(*********************************** G.D S.p.A. - Technical Department ***********************************
============= PROGRAM INFO ============
FOLDER:             TBD
MACHINES INVOLVED:  TBD 

============= DESCRIPTION =============
csp machine declaration

============= REVISIONS ===============
Date		Version	 	Author      	Description             
----------	-------		------------  	--------------------------------------------
2019/04/05 	0000.00	 	M.Grasso		Creation of the PRG

**********************************************************************************************************)
(*$R process_ref := prc; $*)
PROGRAM csp_transfer_infeed_accumulation
VAR
	
	prc:											process;
	prc_path:										STRING;
	
	accumulation_conveyor_running:					BOOL;
	disable_req:									BOOL;
	
	
END_VAR

_read_var_input();

_object_manager();

IF NOT objects_running()
THEN
	RETURN;	
END_IF

_read_process_image();

_mode_manager();

CASE process_get_mode(prc) OF
	MODE_ABSENT,
	MODE_INACTIVE:
		RETURN;
	MODE_TEST:
		_handle_process_test();
END_CASE


_set_runtime_properties();

(********************************* BODY *********************************)
(************************************************************************)

accumulation_conveyor_running := axis_is_moving(csp_transfer_infeed_accumulation_belt.axis);

disable_req := NOT
				((
				csp_transfer_infeed.run_infeed_belts
				)
				AND
				process_is_ready(prc)
				AND
				process_subtree_is_ready(prc));


_handle_messages();

_write_output();

ACTION _handle_messages:
;
END_ACTION

ACTION _handle_process_test:
;
END_ACTION

ACTION _mode_manager:
IF process_mode_req_is_pending(prc)
THEN
    process_apply_mode_req_first_step(prc);
    CASE process_get_mode(prc) OF
        MODE_TO_ABSENT:
			;
        MODE_TO_INACTIVE:
			;
        MODE_TO_TEST:
			;
        MODE_TO_OPERATIONAL:
			;
    END_CASE
    process_apply_mode_req_second_step(prc);
END_IF
END_ACTION

ACTION _object_manager:
IF objects_initialization()
THEN
	sub_process_init(
		object_name					:= 'csp_transfer_infeed_accumulation.prc', 
		process						:= csp_transfer_infeed.prc, 
		CONVERSION_this				:= prc);
		
	prc_path 						:= process_get_path(prc);
	
END_IF

IF objects_running()
THEN
	process_cycle(prc);
END_IF
END_ACTION

ACTION _read_process_image:
;
END_ACTION

ACTION _read_var_input:
;
END_ACTION

ACTION _set_runtime_properties:
;
END_ACTION

ACTION _write_output:
;
END_ACTION

END_PROGRAM

(* stored: Version 1.1.0.1, ProductVersion 3.1.4024.3
   POU csp_transfer_infeed_accumulation: Id {a79cd134-3646-4220-9711-3f94c224ec2d}, SpecialFunc None
   Action _handle_messages: Id {b79f2d6d-428a-4ddf-8301-7fd94ca80f10}
   Action _handle_process_test: Id {f858689f-18b2-4f51-95e1-907e4326fa7a}
   Action _mode_manager: Id {b55a7ea0-3679-46bc-808b-ce3e5b871f1a}
   Action _object_manager: Id {b710be2e-cae6-4a98-aabe-a7a491602cc1}
   Action _read_process_image: Id {25411fa8-82f9-44ef-8b06-06fcb17cdc8b}
   Action _read_var_input: Id {5b4e7ba7-7a10-4636-91ef-676858d06c97}
   Action _set_runtime_properties: Id {bcffe2bd-b772-4b09-906f-098d2b4dbc94}
   Action _write_output: Id {81e35ab2-eb56-4080-9d7c-8a6886c23a4c} *)
